INTERFACE ITF_BaseExecutiveElement

END_INTERFACE

(* stored: Version 1.1.0.1
   Itf ITF_BaseExecutiveElement: Id {ad3f64dc-ad28-0928-11ba-a3b4f43ec05a} *)
